PROGRAM MAIN
VAR
	bIn : BOOL;
	bOut : BOOL;
END_VAR

bIn := GVL.bIn;

GVL.bOut := bOut;

END_PROGRAM

(* stored: Version 1.1.0.1, ProductVersion 3.1.4024.12
   POU MAIN: Id {1c5099ca-8ba9-4952-97a3-dfd211cf5f06}, SpecialFunc None *)
